INTERFACE I_HostParameters EXTENDS __SYSTEM.IQueryInterface

PROPERTY Parameters : I_Parameters
GET
END_GET
END_PROPERTY

END_INTERFACE

(* stored: Version 1.1.0.1, ProductVersion 3.1.4024.12
   Itf I_HostParameters: Id {d0522bc1-9686-4532-9647-ae9732b4bf43}
   Property Parameters: Id {fcb4c504-d0fc-498a-a39a-8f84628064d8}
   Get Get: Id {2532a93a-3fe7-4b04-b285-063a230e388c} *)
